// This function has been automatically generated from the project information.
{attribute 'signature_flag' := '1073741824'}
{attribute 'TcGenerated'}
{attribute 'no-analysis'}
FUNCTION F_GetTitle : WSTRING
VAR_INPUT
	
END_VAR

F_GetTitle := "TAC_Events";

END_FUNCTION

(* stored: Version 1.1.0.1, ProductVersion 3.1.4026.12
   POU F_GetTitle: Id {c920a547-f02e-411e-83ee-95cd6186cd26}, SpecialFunc None *)
